// TIA Portal V20 export
// export: Created 2026-04-11T06:02:29.9324966Z, ExportSetting WithDefaults, DisplayName Totally Integrated Automation Portal, DisplayVersion V20, DisplayName TIA Portal Openness, DisplayVersion V20, DisplayName TIA Portal Version Control Interface, DisplayVersion V20, DisplayName STEP 7 Professional, DisplayVersion V20, DisplayName STEP 7 Safety, DisplayVersion V20, DisplayName WinCC Basic/Comfort/Advanced, DisplayVersion V20, DisplayName WinCC Unified, DisplayVersion V20
TYPE "udtError_AnalogOutput"
// stored: IsFailsafeCompliant false
   STRUCT
      OutOfRange { ExternalWritable := 'False'} : Bool;   // Input value is outside range of engineering units
      ConfigurationError { ExternalWritable := 'False'} : Bool;   // Engineering units are not properly configured
   END_STRUCT;
END_TYPE
